// TIA Portal project "Bulat_course_project" (V16)

(* hardware
DEVICE "S7-1200 station_1"  S7-1200 Station
   slot 0: "Rack_0"  S7-1200 Rack  Rack  V1.0
   slot 1: "PLC_1"  CPU 1215C AC/DC/Rly  6ES7 215-1BG40-0XB0  V4.4
DEVICE "CSM"  SCALANCE X-Station
   slot 0: "SCALANCE X rack"  Rail
   slot 0: "Switch_1"  6GK7 277-1AA10-0AA0
DEVICE "HMI_1"  KTP700 Basic PN
   slot 0: "HMI_1"  KTP700 Basic PN  6AV2 123-2GB03-0AX0  15.1.0.0
   slot 1: "HMI_RT_1"  KTP700 Basic PN  6AV2 123-2GB03-0AX0  15.1.0.0
   slot 5: "HMI_1.IE_CP_1"  PROFINET Interface  15.0.1.0
      slot 1: "PROFINET Interface_1"  PROFINET Interface
         slot 1: "Port_1"  Port
*)

// ===== PLC "PLC_1"  CPU 1215C AC/DC/Rly =====

VAR_GLOBAL   // PLC tag table "Process"
   "process_bar_70" AT %QW0 : Int;
END_VAR

ORGANIZATION_BLOCK "Main"   // OB1, LAD, ProgramCycle
TITLE = "Main Program Sweep (Cycle)"
{ S7_Optimized_Access := 'TRUE' }
VERSION : 0.1
   VAR_INPUT
      Initial_Call : Bool;   // Initial call of this OB
      Remanence : Bool;   // =True, if remanent data are available
   END_VAR
BEGIN
END_ORGANIZATION_BLOCK

(* ===== HMI "HMI_RT_1" =====
connection "HMI_Connection_1": ETHERNET, SMART_S7_1200_OMS

HMI tags "Default tag table"
   "process_bar_70" : Int = PLC process_bar_70 AT %QW0, 1 s

screen "Main_Page" 800x480
   GraphicView "Graphic view_38" at 157,407 size 15x15; Picture "Graphic_21"
   GraphicView "Graphic view_39" at 172,406 size 15x15; Picture "Graphic_22"
   GraphicView "Graphic view_40" at 158,279 size 15x15; Picture "Graphic_21"
   GraphicView "Graphic view_41" at 173,278 size 15x15; Picture "Graphic_22"
   GraphicView "Graphic view_42" at 265,279 size 15x15; Picture "Graphic_21"
   GraphicView "Graphic view_43" at 280,278 size 15x15; Picture "Graphic_22"
   GraphicView "Graphic view_44" at 381,279 size 15x15; Picture "Graphic_21"
   GraphicView "Graphic view_45" at 396,278 size 15x15; Picture "Graphic_22"
   GraphicView "Graphic view_46" at 488,279 size 15x15; Picture "Graphic_21"
   GraphicView "Graphic view_47" at 503,278 size 15x15; Picture "Graphic_22"
   GraphicView "Graphic view_48" at 264,134 size 15x15; Picture "Graphic_21"
   GraphicView "Graphic view_49" at 279,133 size 15x15; Picture "Graphic_22"
   GraphicView "Graphic view_50" at 381,134 size 15x15; Picture "Graphic_21"
   GraphicView "Graphic view_51" at 396,133 size 15x15; Picture "Graphic_22"
   GraphicView "Graphic view_52" at 497,134 size 15x15; Picture "Graphic_21"
   GraphicView "Graphic view_53" at 512,133 size 15x15; Picture "Graphic_22"
   GraphicView "Graphic view_54" at 579,134 size 15x15; Picture "Graphic_21"
   GraphicView "Graphic view_55" at 594,133 size 15x15; Picture "Graphic_22"
   GraphicView "Graphic view_56" at 697,139 size 15x15; Picture "Graphic_21"
   GraphicView "Graphic view_57" at 712,138 size 15x15; Picture "Graphic_22"
   GraphicView "Graphic view_58" at 574,274 size 15x15; Picture "Graphic_21"
   GraphicView "Graphic view_59" at 589,273 size 15x15; Picture "Graphic_22"
   GraphicView "Graphic view_60" at 173,186 size 50x23; Picture "Graphic_29"
   Button "Button_1" at 23,107 size 96x32; TextOff 'Start'
   Button "Button_2" at 18,225 size 96x32; TextOff 'Stop'
   GraphicView "Graphic view_1" at 22,424 size 126x56; Picture "Graphic_1"
   GraphicView "Graphic view_2" at 144,374 size 56x97; Picture "Graphic_2"
   GraphicView "Graphic view_4" at 141,4 size 62x70; Picture "Graphic_8"
   GraphicView "Graphic view_3" at 142,67 size 60x332; Picture "Graphic_4"
   GraphicView "Graphic view_6" at 198,3 size 60x70; Picture "Graphic_10"
   GraphicView "Graphic view_5" at 135,210 size 81x113; Picture "Graphic_6"
   GraphicView "Graphic view_7" at 253,3 size 60x70; Picture "Graphic_11"
   GraphicView "Graphic view_9" at 253,169 size 60x56; Picture "Graphic_4"
   GraphicView "Graphic view_8" at 244,68 size 81x113; Picture "Graphic_6"
   GraphicView "Graphic view_10" at 364,169 size 60x57; Picture "Graphic_4"
   GraphicView "Graphic view_11" at 367,4 size 60x70; Picture "Graphic_8"
   GraphicView "Graphic view_12" at 425,3 size 60x70; Picture "Graphic_10"
   GraphicView "Graphic view_13" at 357,68 size 81x113; Picture "Graphic_6"
   GraphicView "Graphic view_14" at 480,3 size 60x70; Picture "Graphic_11"
   GraphicView "Graphic view_15" at 480,169 size 60x57; Picture "Graphic_4"
   GraphicView "Graphic view_16" at 471,68 size 81x113; Picture "Graphic_6"
   GraphicView "Graphic view_17" at 565,174 size 60x54; Picture "Graphic_4"
   GraphicView "Graphic view_18" at 568,9 size 60x70; Picture "Graphic_8"
   GraphicView "Graphic view_19" at 626,8 size 60x70; Picture "Graphic_10"
   GraphicView "Graphic view_20" at 558,73 size 81x113; Picture "Graphic_6"
   GraphicView "Graphic view_21" at 681,8 size 60x70; Picture "Graphic_11"
   GraphicView "Graphic view_22" at 681,174 size 60x149; Picture "Graphic_4"
   GraphicView "Graphic view_23" at 672,73 size 81x113; Picture "Graphic_6"
   GraphicView "Graphic view_24" at 244,210 size 81x113; Picture "Graphic_6"
   GraphicView "Graphic view_25" at 357,209 size 81x113; Picture "Graphic_6"
   GraphicView "Graphic view_26" at 471,210 size 81x113; Picture "Graphic_6"
   GraphicView "Graphic view_27" at 558,210 size 81x113; Picture "Graphic_6"
   GraphicView "Graphic view_29" at 254,318 size 60x70; Picture "Graphic_16"
   GraphicView "Graphic view_30" at 311,318 size 60x70; Picture "Graphic_10"
   GraphicView "Graphic view_31" at 367,318 size 60x70; Picture "Graphic_17"
   GraphicView "Graphic view_32" at 474,318 size 60x70; Picture "Graphic_16"
   GraphicView "Graphic view_33" at 531,318 size 42x70; Picture "Graphic_10"
   GraphicView "Graphic view_34" at 568,318 size 60x70; Picture "Graphic_17"
   GraphicView "Graphic view_35" at 681,318 size 60x70; Picture "Graphic_16"
   GraphicView "Graphic view_36" at 735,318 size 42x70; Picture "Graphic_10"
   Group "Group" at 325,350 size 28x8
   Group "Group_1" at 536,350 size 28x8
   Group "Group_2" at 746,350 size 28x8
   Group "Group_3" at 5,449 size 28x8
   Group "Group_4" at 165,342 size 8x26
   Group "Group_5" at 165,149 size 8x26
   Group "Group_6" at 391,182 size 8x26
   Group "Group_7" at 591,187 size 8x26
   Group "Group_8" at 638,35 size 28x8
   Group "Group_9" at 438,31 size 28x8
   Group "Group_10" at 210,34 size 28x8
   Group "Group_11" at 505,182 size 8x29
   Group "Group_12" at 277,181 size 8x29
   Group "Group_13" at 708,249 size 8x29
   TextField "Text field_1" at 149,250 size 45x23; Text 'K1/3'
   TextField "Text field_2" at 271,107 size 16x23; Text 'X'
   TextField "Text field_3" at 381,107 size 25x23; Text 'Ty'
   TextField "Text field_4" at 497,107 size 16x23; Text 'X'
   TextField "Text field_5" at 574,106 size 32x23; Text 'E-2'
   TextField "Text field_6" at 693,106 size 30x23; Text 'CM'
   TextField "Text field_7" at 265,249 size 26x23; Text 'K2'
   TextField "Text field_8" at 382,249 size 26x23; Text 'K3'
   TextField "Text field_9" at 491,249 size 32x23; Text 'E-1'
   TextField "Text field_10" at 583,249 size 16x23; Text 'X'
   TextField "Text field_11" at 39,440 size 47x20; Text 'Сырьё'
   TextField "Text field_12" at 182,66 size 45x20; Text 'Смесь'
   TextField "Text field_13" at 145,81 size 99x20; Text 'денормализата'
   TextField "Text field_14" at 271,392 size 92x20; Text 'денормализат'
   TextField "Text field_15" at 260,375 size 81x20; Text 'Стабильный'
   TextField "Text field_16" at 470,369 size 45x20; Text 'Смесь'
   TextField "Text field_17" at 470,386 size 94x20; Text 'промывочного'
   TextField "Text field_18" at 469,406 size 62x20; Text 'продукта'
   TextField "Text field_19" at 722,302 size 71x20; Text 'Парафины'
   TextField "Text field_20" at 700,370 size 99x20; Text 'денормализата'
   Group "Group_14" at 157,406 size 30x16; Picture "Graphic_21"
   Group "Group_15" at 158,278 size 30x16; Picture "Graphic_21"
   Group "Group_16" at 265,278 size 30x16; Picture "Graphic_21"
   Group "Group_17" at 381,278 size 30x16; Picture "Graphic_21"
   Group "Group_18" at 488,278 size 30x16; Picture "Graphic_21"
   Group "Group_19" at 264,133 size 30x16; Picture "Graphic_21"
   Group "Group_20" at 381,133 size 30x16; Picture "Graphic_21"
   Group "Group_21" at 497,133 size 30x16; Picture "Graphic_21"
   Group "Group_22" at 579,133 size 30x16; Picture "Graphic_21"
   Group "Group_23" at 697,138 size 30x16; Picture "Graphic_21"
   Group "Group_24" at 574,273 size 30x16; Picture "Graphic_21"
   GraphicView "Graphic view_28" at 110,406 size 25x24; Picture "Graphic_27"
   GraphicView "Graphic view_37" at 180,236 size 27x20; Picture "Graphic_28"
   GraphicView "Graphic view_61" at 305,192 size 25x26; Picture "Graphic_30"
   GraphicView "Graphic view_62" at 425,192 size 25x26; Picture "Graphic_30"
   GraphicView "Graphic view_63" at 439,67 size 25x26; Picture "Graphic_30"
   GraphicView "Graphic view_64" at 539,52 size 25x26; Picture "Graphic_30"

screen "Process_Page" 800x480
   Bar "Bar_1" at 150,122 size 173x246; MinimumValue 0; MaximumValue 100
      ProcessValue <- "process_bar_70"
   Button "Button_1" at 23,107 size 96x32; TextOff 'Start'
   Button "Button_2" at 18,225 size 96x32; TextOff 'Stop'
   IOField "I/O field_1" at 219,37 size 96x32; FormatPattern s9999
      ProcessValue <- "process_bar_70"
   TrendView "Trend view_1" at 344,29 size 452x447
   DateTimeField "Date/time field_1" at 204,417 size 116x32
   TextField "Text field_1" at 140,8 size 177x23; Text 'Давление в колонне'
   TextField "Text field_2" at 207,92 size 75x23; Text 'Уровень'
   TextField "Text field_3" at 398,37 size 198x23; Text 'Показатель изменения'
   TextField "Text field_4" at 198,394 size 68x23; Text 'Таймер'
   Button "Button_3" at 8,404 size 120x64; TextOff 'Main page'
*)